{attribute 'linkalways'} 
{attribute 'no_explicit_call' := 'This FB is a CLASS and must be accessed using methods or properties'}
{attribute 'enable_dynamic_creation'}
FUNCTION_BLOCK _Array0to2OfINT EXTENDS ArrayDatatypeBase_1D
VAR CONSTANT
	lBound : DINT := 0;
	uBound : DINT := 2;
END_VAR
VAR
	localData : ARRAY [lBound..uBound] OF INT;
	activeData : REFERENCE TO ARRAY [lBound..uBound] OF INT REF= localData;
	elements : ARRAY [lBound..uBound] OF _INT(0);
	baseType : _INT(0);
END_VAR

PROPERTY PUBLIC Address : PVOID
GET
Address := ADR(activeData);
END_GET
END_PROPERTY

PROPERTY PUBLIC BaseDatatype : I_Datatype
GET
BaseDatatype := baseType;
END_GET
END_PROPERTY

METHOD PUBLIC ClearReference
VAR_INPUT
END_VAR
activeData REF= localData;
SetElementReference();
END_METHOD

METHOD PUBLIC Clone : I_Datatype
VAR
    pClone : POINTER TO _Array0to2OfINT;
END_VAR
pClone := __NEW(_Array0to2OfINT());
pClone^.Value := Value;
Clone := pClone^;
END_METHOD

METHOD FB_init : BOOL
VAR_INPUT
	bInitRetains : BOOL; // if TRUE, the retain variables are initialized (warm start / cold start)
	bInCopyCode : BOOL;  // if TRUE, the instance afterwards gets moved into the copy code (online change)
END_VAR
SetElementReference();
END_METHOD

METHOD PUBLIC MakeReferenceTo
VAR_INPUT
	ReferenceTarget : REFERENCE TO ARRAY [lBound..uBound] OF INT;
END_VAR
activeData REF= ReferenceTarget;
SetElementReference();
END_METHOD

METHOD PROTECTED OnSerializeArrayValues
VAR_INPUT
	Serializer : I_Serializer;
END_VAR
VAR
	i : DINT;
END_VAR
FOR i := lBound TO uBound DO
	elements[i].SerializeWith(Serializer);
END_FOR
END_METHOD

METHOD PROTECTED SetElementReference
VAR_INPUT
END_VAR
VAR
	i : DINT;
END_VAR
FOR i := lBound TO uBound DO
	elements[i].MakeReferenceTo(activeData[i]);
END_FOR
END_METHOD

PROPERTY PUBLIC Size : UDINT
GET
Size := SIZEOF(activeData);
END_GET
END_PROPERTY

METHOD PROTECTED TryDeserializeArrayValues : BOOL
VAR_INPUT
	Deserializer : I_Deserializer;
	Feedback : I_DeserializerFeedback;
END_VAR
VAR
	enumerator : I_DeserializerArrayForwardEnumerator;
	i : DINT;
END_VAR
enumerator := Deserializer.GetArrayEnumerator();
i := lBound;

WHILE enumerator.MoveNext() AND i <= uBound DO
	
	IF NOT elements[i].TryDeserializeFrom(enumerator.Current, Feedback) THEN
		EXIT;
	END_IF
	i := i + 1;

END_WHILE
enumerator.Dispose();
END_METHOD

METHOD PUBLIC TryGetElementAsDatatypeByIndex : BOOL
VAR_INPUT
	Index : DINT;
	Destination : REFERENCE TO I_Datatype;
END_VAR
IF Index < lbound OR Index > ubound THEN
	RETURN;
END_IF

Destination := elements[Index];
TryGetElementAsDatatypeByIndex := TRUE;
END_METHOD

METHOD PUBLIC TryGetLowerBound : BOOL
VAR_INPUT
	Dimention : UDINT;
	Destination : REFERENCE TO DINT;
END_VAR
IF Dimention = 1 THEN
	Destination := lBound;
	TryGetLowerBound := TRUE;
END_IF
END_METHOD

METHOD PUBLIC TryGetUpperBound : BOOL
VAR_INPUT
	Dimention : UDINT;
	Destination : REFERENCE TO DINT;
END_VAR
IF Dimention = 1 THEN
	Destination := uBound;
	TryGetUpperBound := TRUE;
END_IF
END_METHOD

METHOD TryMakeReferenceTo : BOOL
VAR_INPUT
	Target : I_Datatype;
END_VAR
VAR
	pTargetData : POINTER TO ARRAY [lBound..uBound] OF INT;
END_VAR
IF NOT IsEquivalentTo(Target) THEN
	RETURN;
END_IF

pTargetData := Target.Address;
activeData REF= pTargetData^;
SetElementReference();
TryMakeReferenceTo := TRUE;
END_METHOD

PROPERTY PUBLIC Value : REFERENCE TO ARRAY [lBound..uBound] OF INT;
GET
Value ref= activeData;
END_GET
END_PROPERTY

END_FUNCTION_BLOCK

(* stored: Version 1.1.0.1, ProductVersion 3.1.4024.13
   POU _Array0to2OfINT: Id {1959a93f-cc9f-0342-0ebe-5a793ff3cf19}, SpecialFunc None
   Folder Core: Id {395f4dd0-0d56-08d5-2c25-36532ad5b650}
   Folder Constructor: Id {1191f26c-67f3-09ab-2c9f-14a1da11c1dd}
   Folder Protected: Id {2ed9423b-ddda-0de0-22e1-73c5fc8ef9ff}
   Folder Customize: Id {650e5166-351f-0dc8-10fa-a7a9da1f4319}
   Property Address: Id {a60d20b1-1411-0ede-2262-816b4fb15d99}
   Get Get: Id {fe3d5874-aef1-040b-0352-4ae35945e2f0}
   Property BaseDatatype: Id {c18f0616-1dc0-0873-3997-4d856c96dce9}
   Get Get: Id {8d520879-640b-0798-383c-f8005d897cdb}
   Method ClearReference: Id {d3b98aad-8f6c-0990-2bcb-4b1ea2ea4882}
   Method Clone: Id {5d2cc844-18d8-0fa7-032e-d08b3e0f1b34}
   Method FB_init: Id {346c4eaa-578b-0331-2ad8-cd7740cfcf86}
   Method MakeReferenceTo: Id {57ea10b3-d3cb-0cbe-2c20-9e7b23a28d43}
   Method OnSerializeArrayValues: Id {1c76b51d-2813-0075-0c1a-0555bfd1d4e8}
   Method SetElementReference: Id {3ee4d691-b5dd-031f-3725-c586ae3adf85}
   Property Size: Id {21a51318-4117-0d5d-36bf-d014e4e5a8d9}
   Get Get: Id {0a11c282-c9c0-024d-3a0e-e7caea331a0f}
   Method TryDeserializeArrayValues: Id {cd3fd1ad-6a31-00be-338a-575c330de77c}
   Method TryGetElementAsDatatypeByIndex: Id {080200c5-ec0a-0d8f-0f79-183339155172}
   Method TryGetLowerBound: Id {2e134cc9-240c-0cf7-1e71-8745db99d456}
   Method TryGetUpperBound: Id {0616d0b6-0cb5-087d-2a6f-75c9064a2c25}
   Method TryMakeReferenceTo: Id {2466093a-0f02-0eef-235d-20f2ec21ee25}
   Property Value: Id {dd9572d4-b23a-0091-071b-193e0e11bd62}
   Get Get: Id {94db1897-4f69-0910-32fa-1c1c799f1e10} *)
